// TIA Portal V20 export
// export: Created 2025-12-01T14:57:10.7856066Z, ExportSetting None, DisplayName Totally Integrated Automation Portal, DisplayVersion V20 Update 3, DisplayName TIA Portal Openness, DisplayVersion V20 Update 3, DisplayName TIA Portal Version Control Interface, DisplayVersion V20 Update 3, DisplayName STEP 7 Professional, DisplayVersion V20 Update 3, DisplayName STEP 7 Safety, DisplayVersion V20 Update 2, DisplayName WinCC Basic/Comfort/Advanced, DisplayVersion V20 Update 3, DisplayName WinCC Professional, DisplayVersion V20 Update 3, DisplayName WinCC Unified, DisplayVersion V20 Update 3
FUNCTION "FC827_CalcularOrdenUT_MesaMultiDestino" : Void   // FC827, STL
{ S7_Optimized_Access := 'FALSE' }
// stored: AutoNumber false
   VAR_INPUT
      NumeroUT : UInt;
   END_VAR
   VAR_OUTPUT
      Orden : Word;   // Orden a realizar en la MESA
      Auxiliar_01 : UInt;   // Auxiliar 01 de la Orden a realizar en la MESA
      MesaSalidaMulti : UInt;   // Auxiliar 02 de la Orden a realizar en la MESA
      Auxiliar_03 : UInt;   // Auxiliar 03 de la Orden a realizar en la MESA
      Auxiliar_04 : UInt;   // Auxiliar 04 de la Orden a realizar en la MESA
   END_VAR
   VAR_TEMP
      IndiceMesaSalida : UInt;
      DatosMesaOrigen : UInt;
      DatosMesaDestino : UInt;
      DatosMesaSalida : UInt;
      P_Temporal : DWord;
      MesaOrigenUT : UInt;
      MesaDestinoUT : UInt;
      MesaIntermediaUT : UInt;
      NumeroMesa : UInt;
      SiguienteUT : UInt;
      OrdenTMP : Word;
      ValorReturn : Int;
      SinUT_EnMesa : Bool;
      RutaOK_EnMesa : Bool;
   END_VAR
BEGIN

NETWORK
TITLE = Inicializar
/////////////////////////////////////////////////////////////////////////
// Inicializaciones de las variables de los DB's

      L     0;
      T     #Orden;
      T     #OrdenTMP;
      T     #MesaSalidaMulti;
      T     #Auxiliar_01;
      T     #Auxiliar_03;
      T     #Auxiliar_04;


/////////////////////////////////////////////////////////////////////////
// Mesa Actual dentro del PLC
      L     "DB812_UTs_Control".UT[#NumeroUT].MesaActual;
      L     "CTE_OffsetMesa";
      -I;
      T     #NumeroMesa;



NETWORK
TITLE = Calcular Orden - FASE 01 >>> Busqueda de la Mesa de Salida
/////////////////////////////////////////////////////////////////////////
// --- Es una Mesa de Multiple Destinos      NUEVA OPERATIVA   14/10/2014
/////////////////////////////////////////////////////////////////////////
// ---
// --- Se realizará lo siguiente:
// --- * Verificacion de que la mesa destino esta libre
// --- * Se enviara la orden por defecto
// --- * Auxiliar_02 = Mesa Intermedia
// --- * Dar por tratada
// --- * Recoger la siguiente mesa de la RUTA
// ---
/////////////////////////////////////////////////////////////////////////


/////////////////////////////////////////////////////////////////////////
/////////////////////////////////////////////////////////////////////////
/////////////////////////////////////////////////////////////////////////
// FASE 01 >>> Calcular la Mesa de Salida


/////////////////////////////////////////////////////////////////////////
// 1 >>> Mesa Origen de la Busqueda
      L     "DB812_UTs_Control".UT[#NumeroUT].MesaActual;
      L     "CTE_OffsetMesa";
      -I;
      T     #MesaOrigenUT;


/////////////////////////////////////////////////////////////////////////
// 2 >>> Mesa Destino de la Busqueda
      L     "DB812_UTs_Control".UT[#NumeroUT].MesaDestino;
      L     "CTE_OffsetMesa";
      -I;
      T     #MesaDestinoUT;


/////////////////////////////////////////////////////////////////////////
// 3 >>> Realizar Busqueda

      L     0;
      T     #IndiceMesaSalida;
InicioBucleBusqueda_MesaSalida:NOP   0;


/////////////////////////////////////////////////////////////////////////
// 3.1 >>> Recoger datos
      L     "DB851_SalidaMesaMultiplesDestinos".MesaSalida[#IndiceMesaSalida].Origen;
      T     #DatosMesaOrigen;
      L     "DB851_SalidaMesaMultiplesDestinos".MesaSalida[#IndiceMesaSalida].Destino;
      T     #DatosMesaDestino;
      L     "DB851_SalidaMesaMultiplesDestinos".MesaSalida[#IndiceMesaSalida].Intermedia;
      T     #DatosMesaSalida;


/////////////////////////////////////////////////////////////////////////
// 3.2 >>> Controles de los datos de la Lista de Mesas de Salida
      L     #DatosMesaOrigen;
      L     0;
      ==I;  // Final de la Lista ?
      JC    FinalBucleBusqueda_MesaSalida;

      L     #DatosMesaOrigen;
      L     #MesaOrigenUT;
      <>I;  // Mesa Origen encontrada ?
      JC    ContinuarBucleBusqueda_MesaSalida;

      L     #DatosMesaDestino;
      L     #MesaDestinoUT;
      <>I;  // Mesa Destino encontrada ?
      JC    ContinuarBucleBusqueda_MesaSalida;


/////////////////////////////////////////////////////////////////////////
// 3.3 >>> Encontrada, en "DatosMesaSalida" estan los Datos
      JU    FinalBucleBusqueda_MesaSalida;


/////////////////////////////////////////////////////////////////////////
// 3.4 >>> No Encontrado pasar a la siguiente de la lista
ContinuarBucleBusqueda_MesaSalida:NOP   0;
      L     #IndiceMesaSalida;
      L     1;
      +I;
      T     #IndiceMesaSalida;

      JU    InicioBucleBusqueda_MesaSalida;


/////////////////////////////////////////////////////////////////////////
// 4 >>> Final del Bucle De Busqueda -  Final de FASE 01
//       Hay Posible destino
FinalBucleBusqueda_MesaSalida:NOP   0;



NETWORK
TITLE = Calcular Orden - FASE 02 >>> Tiene Libre el Camnino
/////////////////////////////////////////////////////////////////////////
/////////////////////////////////////////////////////////////////////////
/////////////////////////////////////////////////////////////////////////
// FASE 02 >>> Verificar si tiene el camino libre


/////////////////////////////////////////////////////////////////////////
// 1 >>> Existe Mesa de Salida

      L     #DatosMesaSalida;
      L     0;  // No esta Configurada
      ==I;  // Pedir Ruta ?
      JC    PedirRutaNueva_FueraDeRuta;


/////////////////////////////////////////////////////////////////////////
// 2 >>> Verificar que la Mesa de Salida esta Libre

      SET;
      AN    "DB850_DefinicionMesas".Mesa[#NumeroMesa].ConfigMesa.Espera_S01;
      AN    "DB850_DefinicionMesas".Mesa[#NumeroMesa].ConfigMesa.Espera_S02;
      AN    "DB850_DefinicionMesas".Mesa[#NumeroMesa].ConfigMesa.Espera_S03;
      AN    "DB850_DefinicionMesas".Mesa[#NumeroMesa].ConfigMesa.Espera_S04;
      JC    FinalControlEnMesaEspera;

      CALL  "FC870_MesaSinUT"
      ( Mesa  := #DatosMesaSalida,
        SinUT := #SinUT_EnMesa
      );

      SET;  // Mesa esta sin UT ?
      AN    #SinUT_EnMesa;
      JC    FinalCalcularOrden;


/////////////////////////////////////////////////////////////////////////
// 3 >>>> La UT Tiene Camino Libre - Final de FASE 02
FinalControlEnMesaEspera:NOP   0;




NETWORK
TITLE = Calcular Orden - FASE 03 >>> Tiene Ruta Para Continuar
/////////////////////////////////////////////////////////////////////////
/////////////////////////////////////////////////////////////////////////
/////////////////////////////////////////////////////////////////////////
// --- FASE 03, Mirar las rutas de las UT's de la Mesa

      SET;
      A     "DB850_DefinicionMesas".Mesa[#NumeroMesa].ConfigMesa.RutaSalidaTodas;
      O     "DB850_DefinicionMesas".Mesa[#NumeroMesa].ConfigMesa.MultiplesCargasDeSalida;
      O     "DB850_DefinicionMesas".Mesa[#NumeroMesa].ConfigMesa.GrupoDeSalida;
      JCN   FinalControlRutaEnMesa;

      CALL  "FC872_VerificarRutaEnMesa"
      ( Mesa      := #NumeroMesa,
        TestGrupo := "DB850_DefinicionMesas".Mesa[#NumeroMesa].ConfigMesa.GrupoDeSalida,
        RutaOK    := #RutaOK_EnMesa
      );

      SET;  // No tienen todas Ruta ?
      AN    #RutaOK_EnMesa;
      JC    FinalCalcularOrden;

/////////////////////////////////////////////////////////////////////////
// Tiene Ruta para Continuar - Final de FASE 03
FinalControlRutaEnMesa:NOP   0;




NETWORK
TITLE = Calcular Orden - FASE 04 >>> Final, Calcular la Salida de la Mesa
/////////////////////////////////////////////////////////////////////////
/////////////////////////////////////////////////////////////////////////
/////////////////////////////////////////////////////////////////////////
// --- FASE 04, Se envia orden
// --- Primero, doy por tratada la causa
// --- Segundo, Activarse la salida de la mesa

      L     #DatosMesaSalida;
      L     "CTE_OffsetMesa";
      +I;
      T     #MesaIntermediaUT;


/////////////////////////////////////////////////////////////////////////
// 1 >>> Doy por tratada la Mesa la Primera de la Mesa
      L     0;  // Dar por tratada
      T     "DB812_UTs_Control".UT[#NumeroUT].EstadoRecepcionUT;
      T     "DB812_UTs_Control".UT[#NumeroUT].EstadoEventoRecibido;

      L     #MesaIntermediaUT;
      T     "DB812_UTs_Control".UT[#NumeroUT].MesaIntermedia;


/////////////////////////////////////////////////////////////////////////
// 2 >>> Si hay que darla por tratadas todas las de la Mesa

      SET;  // Hay que Recorrer el Resto de UTs de la Mesa
      AN    "DB850_DefinicionMesas".Mesa[#NumeroMesa].ConfigMesa.MultiplesCargasDeSalida;
      AN    "DB850_DefinicionMesas".Mesa[#NumeroMesa].ConfigMesa.GrupoDeSalida;
      JC    FinalBucleUTs_EnMesa;

      L     "DB812_UTs_Control".UT[#NumeroUT].UT_SiguienteMesa;
      T     #SiguienteUT;


InicioBucleUTs_EnMesa:NOP   0;
      L     #SiguienteUT;
      L     0;
      ==I;  // Hay mas UT's
      JC    FinalBucleUTs_EnMesa;

// Testear Grupo ?
      SET;
      AN    "DB850_DefinicionMesas".Mesa[#NumeroMesa].ConfigMesa.GrupoDeSalida;
      JC    ContinuarBucleUTs_EnMesa;

// Dar por tratado solo lo del mismo Grupo
// Grupo Primera UT == Grupo de la Siguiente
      L     "DB812_UTs_Control".UT[#NumeroUT].Grupo;
      L     "DB812_UTs_Control".UT[#SiguienteUT].Grupo;
      <>I;
      JC    FinalBucleUTs_EnMesa;

// Dar por tratada la Siguinete UT
ContinuarBucleUTs_EnMesa:NOP   0;
      L     0;  // Dar por tratada
      T     "DB812_UTs_Control".UT[#SiguienteUT].EstadoRecepcionUT;
      T     "DB812_UTs_Control".UT[#SiguienteUT].EstadoEventoRecibido;

      L     #MesaIntermediaUT;
      T     "DB812_UTs_Control".UT[#SiguienteUT].MesaIntermedia;

      L     "DB812_UTs_Control".UT[#SiguienteUT].UT_SiguienteMesa;
      T     #SiguienteUT;
      JU    InicioBucleUTs_EnMesa;


/////////////////////////////////////////////////////////////////////////
// 2. >>> Final del Bucle
FinalBucleUTs_EnMesa:NOP   0;



/////////////////////////////////////////////////////////////////////////
// 3. >>>  Activarse la salida de la mesa
//         Orden por Defecto
//         Mesa de Salida Multiples Destinos

      L     #DatosMesaSalida;
      T     #MesaSalidaMulti;

      JU    OrdenSalida_Defecto;



NETWORK
TITLE = Control - No existe Mesa de Salida - FUERA de RUTA
/////////////////////////////////////////////////////////////////////////
// --- No existe Mesa de Salida posible
//     La UT esta FUERA de RUTA
//     Realiazar, Evento de Pedir Ruta

PedirRutaNueva_FueraDeRuta:NOP   0;
      L     "DB812_UTs_Control".UT[#NumeroUT].EstadoGeneralUT;
      <>I;  //NO esta LIBRE?
      JC    FinalCalcularOrden;

      L     26;  // 26 - Generar Evento Pedir Ruta (FUERA DE RUTA)
      T     "DB812_UTs_Control".UT[#NumeroUT].EstadoGeneralUT;
      L     0;  // Dar por tratada
      T     "DB812_UTs_Control".UT[#NumeroUT].EstadoRecepcionUT;

      JU    FinalCalcularOrden;



NETWORK
TITLE = Generar Orden de Salida
/////////////////////////////////////////////////////////////////////////
/////////////////////////////////////////////////////////////////////////
// --- Ordenes a enviar dependiendo por donde sale
// --- Salida por S01
OrdenSalida_S01:NOP   0;
      L     P##OrdenTMP;
      L     P#0.1;
      +D;
      T     #P_Temporal;

      SET;  // Orden -> Activar Bit 1
      S     L [#P_Temporal];
      JU    FinalOrdenSalida;


/////////////////////////////////////////////////////////////////////////
/////////////////////////////////////////////////////////////////////////
// --- Ordenes a enviar dependiendo por donde sale
// --- Salida por S02
OrdenSalida_S02:NOP   0;
      L     P##OrdenTMP;
      L     P#0.2;
      +D;
      T     #P_Temporal;

      SET;  // Orden -> Activar Bit 2
      S     L [#P_Temporal];
      JU    FinalOrdenSalida;


/////////////////////////////////////////////////////////////////////////
/////////////////////////////////////////////////////////////////////////
// --- Ordenes a enviar dependiendo por donde sale
// --- Salida por S03
OrdenSalida_S03:NOP   0;
      L     P##OrdenTMP;
      L     P#0.3;
      +D;
      T     #P_Temporal;

      SET;  // Orden -> Activar Bit 3
      S     L [#P_Temporal];
      JU    FinalOrdenSalida;


/////////////////////////////////////////////////////////////////////////
/////////////////////////////////////////////////////////////////////////
// --- Ordenes a enviar dependiendo por donde sale
// --- Salida por S04
OrdenSalida_S04:NOP   0;
      L     P##OrdenTMP;
      L     P#0.4;
      +D;
      T     #P_Temporal;

      SET;  // Orden -> Activar Bit 4
      S     L [#P_Temporal];
      JU    FinalOrdenSalida;



/////////////////////////////////////////////////////////////////////////
/////////////////////////////////////////////////////////////////////////
// --- Ordenes a enviar dependiendo por donde sale
// --- Salida por Defecto
OrdenSalida_Defecto:NOP   0;
      L     P##OrdenTMP;
      L     P#0.5;
      +D;
      T     #P_Temporal;

      SET;  // Orden -> Activar Bit 5
      S     L [#P_Temporal];
      JU    FinalOrdenSalida;


/////////////////////////////////////////////////////////////////////////
/////////////////////////////////////////////////////////////////////////
// No Existen mas posibilidades
FinalOrdenSalida:NOP   0;



NETWORK
TITLE = Final de Calcular Orden
/////////a////////////////////////////////////////////////////////////////
// Finalizar la Funcion
FinalCalcularOrden:NOP   0;

      L     #OrdenTMP;
      T     #Orden;


END_FUNCTION
